Staubli VAL3: remErrBufferGet.pgx

program remErrBufferGet(string& sReturn[] (dimensions=1))
begin
  //Get one error from the error buffer, if there is an error
  //
  logMsg("call remErrBufferGet")
  if sErrBuffer[nErrNow]==""
    sReturn="NOERROR"
  else
    sReturn="ERROR "+sErrBuffer[nErrNow]
    putln(sReturn)
    logMsg(sReturn)
    sErrBuffer[nErrNow]=""
    if nErrNow==nErrBufferSize
      nErrNow=0
    else
      nErrNow=nErrNow+1
    endIf
  endIf
end
